// TIA Portal project "S71200_OPCUA" (V16)

(* hardware
DEVICE "S7-1200 station_1"  S7-1200 Station
   slot 0: "Rack_0"  S7-1200 Rack  Rack  V1.0
   slot 1: "PLC_1"  CPU 1214C DC/DC/Rly  6ES7 214-1HG40-0XB0  V4.4
*)

// ===== PLC "PLC_1"  CPU 1214C DC/DC/Rly =====

DATA_BLOCK "UAServer"   // DB2
{ S7_Optimized_Access := 'TRUE' }
VERSION : 0.1
   VAR
      Start : Bool;
      Led : Bool;
   END_VAR
BEGIN
END_DATA_BLOCK

ORGANIZATION_BLOCK "Main"   // OB1, LAD, ProgramCycle
TITLE = "Main Program Sweep (Cycle)"
{ S7_Optimized_Access := 'TRUE' }
VERSION : 0.1
   VAR_INPUT
      Initial_Call : Bool;   // Initial call of this OB
      Remanence : Bool;   // =True, if remanent data are available
   END_VAR
BEGIN

REGION Network 1
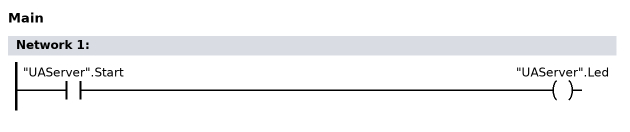
   RUNG wire#powerrail
      Contact( "UAServer".Start )
      Coil( "UAServer".Led )
   END_RUNG
   // the same network as SCL:
   "UAServer".Led := "UAServer".Start;
END_REGION
END_ORGANIZATION_BLOCK

// folder: LGF/7 Signal generators

FUNCTION_BLOCK "LGF_SinusCI"   // FB10027, SCL
TITLE = LGF_SinusCI
{ S7_Optimized_Access := 'TRUE' }
AUTHOR : Siemens_Industry_Support
FAMILY : LGF
NAME : LGF_SinusCI
// This function generates a sinusoidal signal profile. For this it uses the time interval of the calling Cyclic Interrupt OB. / Diese Funktion generiert einen Sinus förmigen Signalverlauf. Er verwendet dazu den Zeittakt des aufrufenden Cyclic Interrupt OB.
   VAR_INPUT
      amplitude : Real := 1.0;   // Amplitude of the signal profile. / Amplitude des Signalverlaufs.
      offset : Real;   // Offset of the signal profile in the Y-direction. / Verschiebung des Signalverlaufs in Y-Richtung.
      periode : UDInt := 1000;   // Period duration of the signal profile in [ms] / Periodendauer des Signalverlaufs in [ms]
      phaseShift : Real;   // Phase offset in [ms] / Phasenverschiebung in [ms]
      callOB : OB_Cyclic;   // Calling cyclic interrupt OB / Aufrufender Weckalarm-OB (Cyclic Interrupt OB)
      reset : Bool;   // Reset of the signal profile. / Rücksetzen des Signalverlaufs.
   END_VAR
   VAR_OUTPUT
      value : Real;   // Current value of the sinusoidal signal. / Aktueller Wert des Sinussignales.
      error : Bool;   // FALSE: No error TRUE: An error occurred during the execution of the FB / FALSE: Kein Fehler TRUE: Während der Ausführung des FB ist ein Fehler aufgetreten
      status : Word;   // 16#0000-16#7FFF: Status of the FB 16#8000-16#FFFF: Error identification (see following Table) / 16#0000-16#7FFF: Status des FB 16#8000-16#FFFF: Fehleridentifikation (siehe folgende Tabelle)
      subFunctionStatus : Word;   // Status or return value of called FB's, FC's and system blocks / Status oder Rückgabewert von aufgerufenen FB's / FC's und Systemfunktionen
   END_VAR
   VAR
      statRad : Real;   // Angle in radians / Size of an angle in radians
      statCounter : UDInt;   // Static Counter value
   END_VAR
   VAR_TEMP
      tempCycleTime : UDInt;   // Temp cycle time from CallOB
      tempCyclePhase : UDInt;   // Temp cycle phase from CallOB
      tempCycleStatus : Word;   // Temp cycle status from CallOB
      tempReadTimeStatus : Int;   // Temp return value of QRY_CINT
   END_VAR
   VAR CONSTANT
      SECOND_IN_MS : UDInt := 1000;   // One second written in miliseconds. Needed in calculation in formulas
      ZERO : Int := 0;   // Numeric zero value
      SLOPE : Int := 2;   // Part of the formula
      TWO_PI : Real := 6.283185;   // 2*PI = ~6.14 / 2*PI = ~6,14
      SUB_STATUS_NO_ERROR : Word := 16#0000;   // Subfunction status: No error
      STATUS_FINISHED_NO_ERROR : Word := 16#0000;   // Status: Execution finished without errors / Status: Abarbeitung ohne Fehler beendet
      QRY_CINT_OB_UNAVAILABLE : Word := 16#0000;   // Cyclic interrupt status: OB not available
      ERR_OB_UNAVAILABLE : Word := 16#8600;   // Error: OB on input `callOB` is not configured / present. Interconnect the constant name of a configured cyclic interrupt OB at the input `callOB`. / Fehler: OB am Eingang `callOB` ist nicht projektiert / vorhanden. Verschalten Sie am Eingang `callOB` den Konstanten Namen eines projektierten Weckalarm-OB.
      ERR_QRY_CINT : Word := 16#8601;   // Error in `QRY_CINT` command - check `subFunctionStatus` code / Fehler in Anweisung `QRY_CINT` - weitere Infos in `subFunctionStatus`
   END_VAR
BEGIN
   REGION Block info header
     //===============================================================================
     // SIEMENS AG / (c)Copyright 2019
     //-------------------------------------------------------------------------------
     // Title:            LGF_SinusCI
     // Comment/Function: This function generates a sinusoidal signal profile. For this it uses the time interval of the calling Cyclic Interrupt OB.
     // Library/Family:   LGF (Library General Functions)
     // Author:           Siemens Digital Industry Support
     // Tested with:      CPU 1515F-2 PN FW:V2.6
     // Engineering:      TIA Portal V15.1 Update 2
     // Restrictions:     ENO disabled - error handling done by error and status
     // Requirements:     PLC (S7-1200 / S7-1500)
     //-------------------------------------------------------------------------------
     // Change log table:
     // Version  | Date       | Expert in charge       | Changes applied
     //----------|------------|------------------------|------------------------------
     // 01.00.00 03.07.2018  Siemens Industry Online Support
     //                      First released version
     // 01.00.01 17.08.2018  Siemens Industry Online Support
     //                      Upgrade: TIA V15 Update 2
     // 01.00.02 23.11.2018  Siemens Industry Online Support
     //                      Upgrade: TIA V15.1
     // 01.00.03 26.09.2019  Simatic Systems Support
     //                      Code refactoring, regions and more comments added
     //                      phase shift availability added
     // 03.00.00 23.04.2020  Simatic Systems Support
     //                      Set version to V3.0.0, harmonize the version of the whole library
     // 03.00.01 15.02.2021  Simatic Systems Support
     //                      Insert documentation
     //=============================================================================
   END_REGION Block info header

   REGION DESCRIPTION
     (/*NOTE
   :    The status of called commands is output in `subFunctionStatus`. In this case, the output value in `status` indicates which command caused the error. In this case, refer to the TIA Portal Online Help section for information on the respective commands.

   ---

   The block calculates the values for a sinusoidal signal profile, which is output to the output parameter `value`.

   The `amplitude`, the `offset` in the Y-direction, the `period`, and the `phase shift` can be set at the input parameters.

   The input parameter `reset` resets the signal profile. At the `value` output parameter, the value `0` is output as long as `reset` is set to `TRUE`.

   The block must be called in a cyclic interrupt OB. The time interval of the calling cyclic interrupt OB is determined in the FB with the command `QRY_CINT`. For this, the constant name of the calling cyclic interrupt OB must be interconnected at the input parameter `callOB`.

   ![Interconnecting the cyclic interrupt OB](LGF_InterruptObAsParameter.png "Interconnecting the cyclic interrupt OB")

   The number of calculated values of the signal profile per period duration is calculated as follows:

   $$
     Quantity Values = \frac{Period duration}{Time intervak Cyclic interrupt OB}
   $$

   ---

   Note
   :    To obtain a continuous signal profile of the curve, the time interval of the cyclic interrupt OB should not be selected too large depending on the period duration.

   ---

   ------

   The Figure below shows the signal profile of the calculated values.

   ![LGF_SinusCI](LGF_SinusCI.png "LGF_SinusCI")
   Hinweis
   :    In `subFunctionStatus` wird der Status von aufgerufenen Anweisungen ausgegeben. Der Ausgangswert in `status` gibt in diesem Fall an, welche Anweisung den Fehler verursacht hat. Holen Sie sich in diesem Fall die Informationen aus der TIA Portal Online Hilfe zu den jeweiligen Anweisungen.

   ---

   Der Baustein berechnet die Werte für einen Sinus förmigen Signalverlauf, die am Ausgangsparameter `value` ausgegeben werden.

   Die Amplitude `amplitude`, die Verschiebung in Y-Richtung `offset`, die Periodendauer `periode` und die Phasenverschiebung `phaseShift` können an den Eingangsparametern vorgegeben werden.

   Mit dem Eingangsparameter `reset` wird der Signalverlauf zurückgesetzt. Am Ausgangsparameter `value` wird der Wert `0` ausgegeben, solange `reset` auf `TRUE` gesetzt ist.

   Der Baustein muss in einem Weckalarm-OB (Cyclic Interrupt OB) aufgerufen werden. Der Zeittakt des aufrufenden Weckalarm-OB wird im FB mit der Anweisung `QRY_CINT` ermittelt. Dazu muss am Eingangsparameter `callOB` der Konstanten Name des aufrufenden Weckalarm-OB verschaltet werden.

   ![Weckalarm-OB verschalten](LGF_InterruptObAsParameter.png "Weckalarm-OB verschalten")

   Die Anzahl der berechneten Werte des Signalverlaufs pro Periodendauer errechnet sich folgendermaßen:

   $$
     Anzahl Werte = \frac{Periodendauer}{Zeittakt Weckalarm-OB}
   $$

   ---

   Hinweis
   :    Um einen kontinuierlichen Signalverlauf der Kurve zu erhalten, sollte der Zeittakt des aufrufen Weckalarm-OB in Abhängigkeit von der Periodendauer nicht zu groß gewählt werden.

   ---

   ------

   Die folgende Abbildung zeigt den Signalverlauf der berechneten Werte.

   ![LGF_SinusCI](LGF_SinusCI.png "LGF_SinusCI")*/)
   END_REGION DESCRIPTION

   REGION Get sample time
     // get sample time, according to the cyclic interrupt OB number
     #tempReadTimeStatus := QRY_CINT(OB_NR := #callOB, CYCLE => #tempCycleTime,
                                     PHASE => #tempCyclePhase, STATUS => #tempCycleStatus);

     REGION Error handling
       // Generate error message of the QRY_CINT function
       IF #tempReadTimeStatus <> #ZERO THEN
         #error := TRUE;
         #status := #ERR_QRY_CINT;
         #subFunctionStatus := INT_TO_WORD(#tempReadTimeStatus);
         #value := #ZERO;
         RETURN;

         // Generate error message when OB unavailable
       ELSIF (#tempCycleStatus = #QRY_CINT_OB_UNAVAILABLE) THEN
         #error := TRUE;
         #status := #ERR_OB_UNAVAILABLE;
         #subFunctionStatus := #SUB_STATUS_NO_ERROR;
         #value := #ZERO;
         RETURN;
       END_IF;
     END_REGION
   END_REGION

   REGION Caluclations and outputs assigment
     IF #reset THEN
       #statCounter := 0;
       #value := #ZERO;
     ELSE
       // Increment Counter with each call of "OB_Cyclic_interrupt"
       #statCounter += (#tempCycleTime) / #SECOND_IN_MS;
       #statCounter := #statCounter MOD (#periode);

       // Transfer to radians
       #statRad := UDINT_TO_REAL(#statCounter) * #TWO_PI / (UDINT_TO_REAL(#periode));

       // Calculate output value
       #value := SIN(#statRad + #phaseShift) * #amplitude + #offset;
     END_IF;
     #error := FALSE;
     #status := #STATUS_FINISHED_NO_ERROR;
     #subFunctionStatus := #SUB_STATUS_NO_ERROR;
     //ENO mechanism is not used - forced to true.
     ENO := TRUE;
   END_REGION
END_FUNCTION_BLOCK